Staubli VAL3: remGetMaxV.pgx

program remGetMaxV(string& sReturn[] (dimensions=1))
  local string sCmd
begin
  // Return max translational velocity for remote moves (mm/s)
  //
  logMsg("call remGetMaxV")
  sCmd="GETMAXV"
  call remGetnGlobal(nMaxAccel,sCmd,sReturn)
end
